PROGRAM program1
VAR
	to_2 : INT := 0;
	from_2 : INT := 0;
END_VAR

gvl.from_1_to_2 := to_2;
from_2 := gvl.from_2_to_1;

END_PROGRAM

(* stored: Version 1.1.0.1, ProductVersion 3.1.4024.12
   POU program1: Id {294174a3-fdb4-4db4-8de1-e42c3d8d069a}, SpecialFunc None *)
